PROGRAM MAIN
VAR
END_VAR

END_PROGRAM

(* stored: Version 1.1.0.1
   POU MAIN: Id {62ea0349-62d7-4449-903b-806058a342ed} *)
